// LS Electric XG5000 project: Aula_LS
// PLC LSPLC

PROGRAM Aula_1_05_03_26 (task: Scan Program)

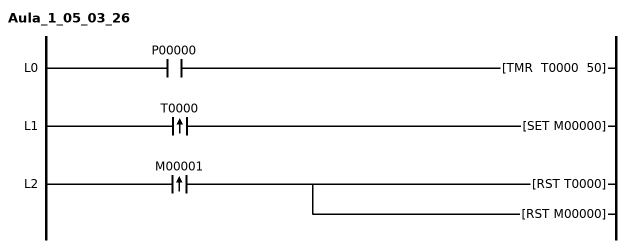
; L0
LOAD      P00000
TMR       T0000 50
; L1
LOADP     T0000
SET       M00000
; L2
LOADP     M00001
RST       T0000
RST       M00000